# EPICS substitutions: ipimbLib/Db/autosave_ipimb.substitutions
#
# ipimb autosave substitutions file
#

# Generate ipimb autosave file
#	Macros:
#		TODO:	List here any macros used in the template
#				Note which ones have defaults.
file autosave_ipimb.template
{
	{
		# Hack till msi supports empty substitutions
		IOC		=	$(IOC),
	}
}
